{attribute 'qualified_only'}
VAR_GLOBAL
	_recipe : stRecipe;
END_VAR

(* stored: Version 1.1.0.1, ProductVersion 3.1.4024.3
   GVL RecipeData: Id {85d83d85-d465-4f76-87be-7e1042ff0a51} *)
